INTERFACE ITF_BaseComponent_HMI_Connector EXTENDS ITF_BaseLoggerElement_HMI_Connector

END_INTERFACE

(* stored: Version 1.1.0.1
   Itf ITF_BaseComponent_HMI_Connector: Id {397afef2-32a5-01a5-03e5-ceebae83b9f0} *)
